TYPE "Coil_Item"
VERSION : 0.1
// Block: Coil_Item
   STRUCT
      C_ID : DInt;
      MES_IDP : String;
      Decoiler_N : Int;
      MES_CN : String;
      MES_HN : String;
      Stato_Rotolo : Int;
      Provini_Richiesti : Int;
      Provini_Eseguiti : Int;
      Diametro_Rotolo : Real;
      Spessore_Errore : Int;
      Spessore_materiale_TAV : Real;
      Spessore_materiale_TEV : Real;
      Spessore_Deroga_TKD : Int;
   END_STRUCT;

END_TYPE
